PROGRAM Test
VAR

	fbTestAlarm1: fbalarm;

	bTes1: BOOL;
	bTest11: BOOL;
	bTestError1: BOOL;
	bTestWarning1: BOOL;
END_VAR

// Door		
	GVL_Status.bSafetyDoorLocked := GVL_Status.bDoorLockCmd;
	GVL_Status.bSafetyDoorUnlocked := GVL_Status.bDoorUnlockCmd;
	
// home
	IF GVL_Status.bHomeCmd THEN
		GVL_Status.bHomeComplete := TRUE;
	END_IF



// Alarm
	fbTestAlarm1(
	bSelectWarning:= bTes1, 
	tDelayTime:= T#1S, 
	bCommand:= TRUE, 
	bAlarmCondition:= bTest11, 
	iAlarmCode:= 1, 
	iPriority:= 1, 
	sAlarmMessage:= 'hello', 
	sLocation:= 'office', 
	bError=> bTestError1, 
	bWarning=> bTestWarning1);

END_PROGRAM

(* stored: Version 1.1.0.1
   POU Test: Id {9e153451-b72e-4319-94b9-29f82d1be8cc}, SpecialFunc None *)
